TYPE ST_PowerMonitor_InputField EXTENDS st_MeasurementVoltageData:
STRUCT
	r_loadshare			: 	REAL;
	Powerlock			: 	ARRAY [1..2] OF ST_MeasurementFieldData;
END_STRUCT
END_TYPE

(* stored: Version 1.1.0.1, ProductVersion 3.1.4024.12
   DUT ST_PowerMonitor_InputField: Id {9360fa12-e620-4f46-a1bd-2737abbc0f8d} *)
